{attribute 'enable_dynamic_creation'}
FUNCTION_BLOCK CMD_Beep IMPLEMENTS I_Command
VAR_INPUT
END_VAR
VAR_OUTPUT
END_VAR
VAR
	Comms : I_CommsTransmitter;
	Status : (IDLE, EXECUTE, SENDING, SENT, COMPLETE, TIMED_OUT);
	WatchDog : WatchDog; 
END_VAR
VAR CONSTANT
	CMD : STRING := 'SYSTem:BEEPer$R$N';
	TIME_OUT : TIME := T#2S;	
END_VAR

CASE Status OF
	
	EXECUTE: 
		WatchDog.Enable(TIME_OUT);
		Status := SENDING;
		
	SENDING:
		IF Comms.isBusy THEN
			RETURN;
		ELSE
			Comms.Send(CMD);
			Status := SENT;
		END_IF
		
	SENT:
		IF Comms.isBusy THEN
			RETURN;
		ELSE
			WatchDog.Disable();
			Status := COMPLETE;
		END_IF
		
	IDLE: //
	COMPLETE://
	TIMED_OUT: //
	
END_CASE

IF WatchDog.isTriggered THEN
	WatchDog.Disable();
	Status := TIMED_OUT;
END_IF

METHOD Destroy
VAR_INPUT
END_VAR
VAR
	selfPointer: POINTER TO CMD_Beep;
END_VAR
selfPointer := ADR(THIS^);
__DELETE(selfPointer);
END_METHOD

METHOD PUBLIC Execute : BOOL
VAR_INPUT

END_VAR
IF NOT isBusy THEN
	Status := EXECUTE;
	Execute := TRUE;
END_IF

THIS^();
END_METHOD

METHOD FB_init : BOOL
VAR_INPUT
	bInitRetains : BOOL; // if TRUE, the retain variables are initialized (warm start / cold start)
	bInCopyCode : BOOL;  // if TRUE, the instance afterwards gets moved into the copy code (online change)
	Comms : I_CommsTransmitter;
END_VAR
THIS^.Comms := Comms;
END_METHOD

PROPERTY PUBLIC hasTimedOut : BOOL
GET
hasTimedOut := (Status = TIMED_OUT) ;
END_GET
END_PROPERTY

PROPERTY PUBLIC isBusy : BOOL
GET
isBusy := not (Status = IDLE or Status = COMPLETE or Status = TIMED_OUT);
END_GET
END_PROPERTY

PROPERTY isComplete : BOOL
GET
isComplete := (Status = COMPLETE or Status = TIMED_OUT) ;
END_GET
END_PROPERTY

END_FUNCTION_BLOCK

(* stored: Version 1.1.0.1, ProductVersion 3.1.4024.9
   POU CMD_Beep: Id {ceed3530-ceb8-4b70-b5a6-b920c843e646}, SpecialFunc None
   Method Destroy: Id {dbace7e7-8252-4843-a9f7-1c5664cd4ded}
   Method Execute: Id {25061073-fedb-4893-9e4a-bddecadd276c}
   Method FB_init: Id {974da62a-5d50-4005-bbc5-46fd62486c62}
   Property hasTimedOut: Id {7ba9a105-c1a3-4748-81d1-184033609fd5}
   Get Get: Id {7fc9873e-8b84-49d1-a1bd-aad55d4debc5}
   Property isBusy: Id {c3b3a263-f0c5-4061-ada2-946d993ea3bb}
   Get Get: Id {5bc46bbc-c90c-4de0-9a47-29fb000ff510}
   Property isComplete: Id {2f5ea95f-2aaa-483a-925e-e7b33079cff9}
   Get Get: Id {ef0460e6-7528-4dc8-9342-2b9526ac8f93} *)
